// TIA Portal V18 export
TYPE "RESET"
// stored: IsFailsafeCompliant true
   STRUCT
      Reset : Bool;
   END_STRUCT;
END_TYPE
